(* Logix 5000 project; controller code_tcc vendor 1 type 14 code 106 rev 33.11; software revision 33.01; part 2 of 3 *)
(* tags used below, declared in another part *)
   Inp_Enable : BOOL;
   Ref_Connection : raC_UDT_ModbusClientConnection;
   Ref_Transactions : raC_UDT_ModbusClientTransaction[5];
   Ref_ModbusData : raC_UDT_ModbusClientData;
   Sts_Faulted : BOOL;
   Sts_Overlap : BOOL;
   Sts_Overload : BOOL;
   Wrk_MSGStep : DINT;
   Wrk_Main_Read_Buffer : STR4096;
   Wrk_WrIndex : DINT;
   Wrk_TransIndex : DINT;
   Wrk_TimerIndex : DINT;
   Wrk_ArraySize : DINT;
   Wrk_LastTransaction : DINT;
   Wrk_ClrReqIndex : DINT;
   Wrk_StepLockTimer : TIMER;
   Wrk_InitCompleted : BOOL;
   HMI_Tab : DINT;
   Wrk_tempHMItransaction : DINT;
   Wrk_HMITransactionValid : BOOL;
   wrk_FAL_Addr : CONTROL;
   wrk_LoopIndex : DINT;
   wrk_AddrIndex : DINT;
   HMI : raC_UDT_ModbusClientHMI;
   Wrk_OLindex : DINT;
   Wrk_OverloadStatus : BOOL;
   Wrk_OverlapStatus : BOOL;
(* raC_Opr_NetModbusTCPClient, continued *)

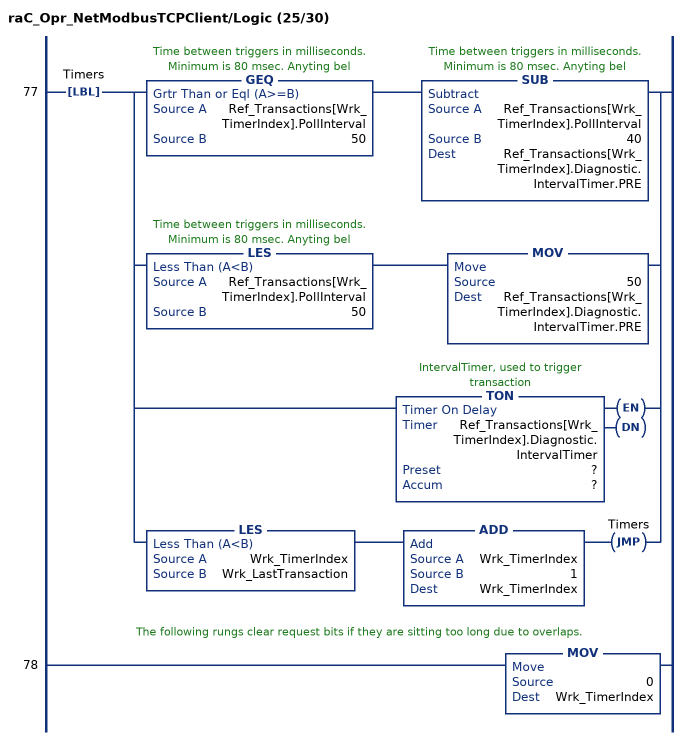
   77: LBL(Timers)[GEQ(Ref_Transactions[Wrk_TimerIndex].PollInterval,50) SUB(Ref_Transactions[Wrk_TimerIndex].PollInterval,40,Ref_Transactions[Wrk_TimerIndex].Diagnostic.IntervalTimer.PRE) ,LES(Ref_Transactions[Wrk_TimerIndex].PollInterval,50) MOV(50,Ref_Transactions[Wrk_TimerIndex].Diagnostic.IntervalTimer.PRE) ,TON(Ref_Transactions[Wrk_TimerIndex].Diagnostic.IntervalTimer,?,?) ,LES(Wrk_TimerIndex,Wrk_LastTransaction) ADD(Wrk_TimerIndex,1,Wrk_TimerIndex) JMP(Timers) ];
   // The following rungs clear request bits if they are sitting too long due to overlaps.
   78: MOV(0,Wrk_TimerIndex);
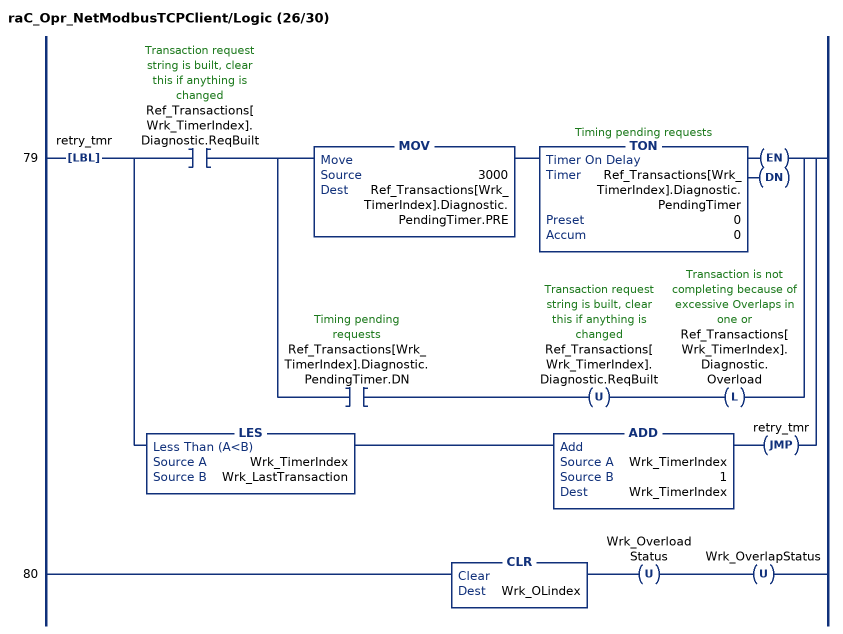
   79: LBL(retry_tmr)[XIC(Ref_Transactions[Wrk_TimerIndex].Diagnostic.ReqBuilt) [MOV(3000,Ref_Transactions[Wrk_TimerIndex].Diagnostic.PendingTimer.PRE) TON(Ref_Transactions[Wrk_TimerIndex].Diagnostic.PendingTimer,0,0) ,XIC(Ref_Transactions[Wrk_TimerIndex].Diagnostic.PendingTimer.DN) OTU(Ref_Transactions[Wrk_TimerIndex].Diagnostic.ReqBuilt) OTL(Ref_Transactions[Wrk_TimerIndex].Diagnostic.Overload) ] ,LES(Wrk_TimerIndex,Wrk_LastTransaction) ADD(Wrk_TimerIndex,1,Wrk_TimerIndex) JMP(retry_tmr) ];
   80: CLR(Wrk_OLindex)OTU(Wrk_OverloadStatus)OTU(Wrk_OverlapStatus);
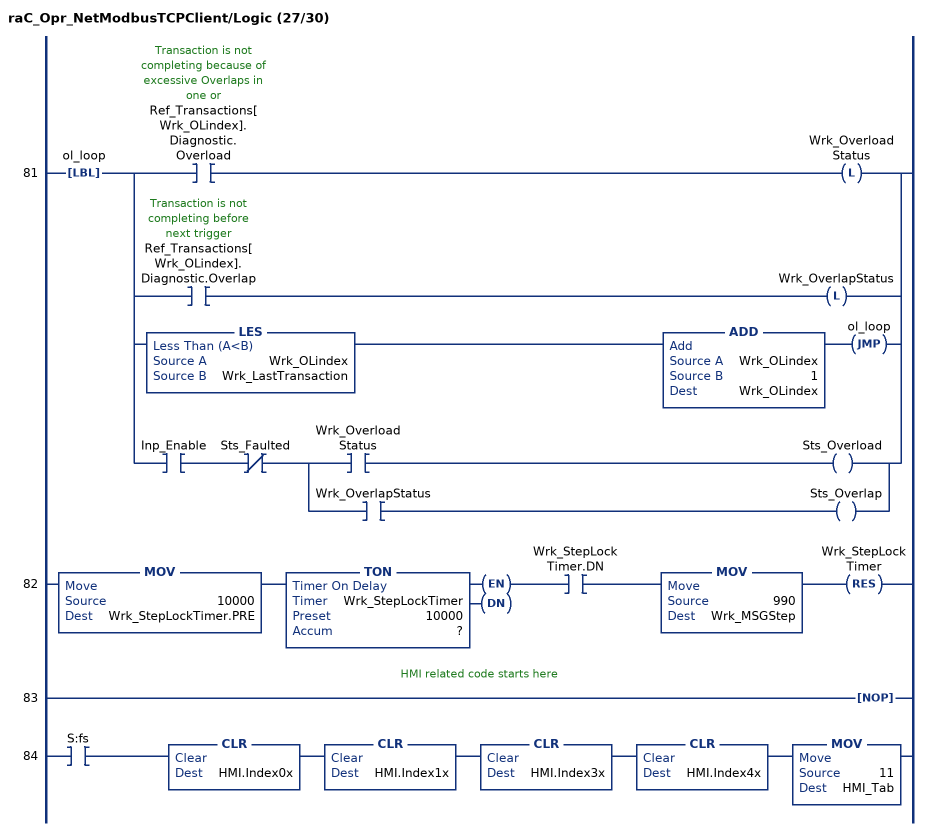
   81: LBL(ol_loop)[XIC(Ref_Transactions[Wrk_OLindex].Diagnostic.Overload) OTL(Wrk_OverloadStatus) ,XIC(Ref_Transactions[Wrk_OLindex].Diagnostic.Overlap) OTL(Wrk_OverlapStatus) ,LES(Wrk_OLindex,Wrk_LastTransaction) ADD(Wrk_OLindex,1,Wrk_OLindex) JMP(ol_loop) ,XIC(Inp_Enable) XIO(Sts_Faulted) [XIC(Wrk_OverloadStatus) OTE(Sts_Overload) ,XIC(Wrk_OverlapStatus) OTE(Sts_Overlap) ] ];
   82: MOV(10000,Wrk_StepLockTimer.PRE)TON(Wrk_StepLockTimer,?,?)XIC(Wrk_StepLockTimer.DN)MOV(990,Wrk_MSGStep)RES(Wrk_StepLockTimer);
   // HMI related code starts here
   83: NOP();
   84: XIC(S:fs)CLR(HMI.Index0x)CLR(HMI.Index1x)CLR(HMI.Index3x)CLR(HMI.Index4x)MOV(11,HMI_Tab);
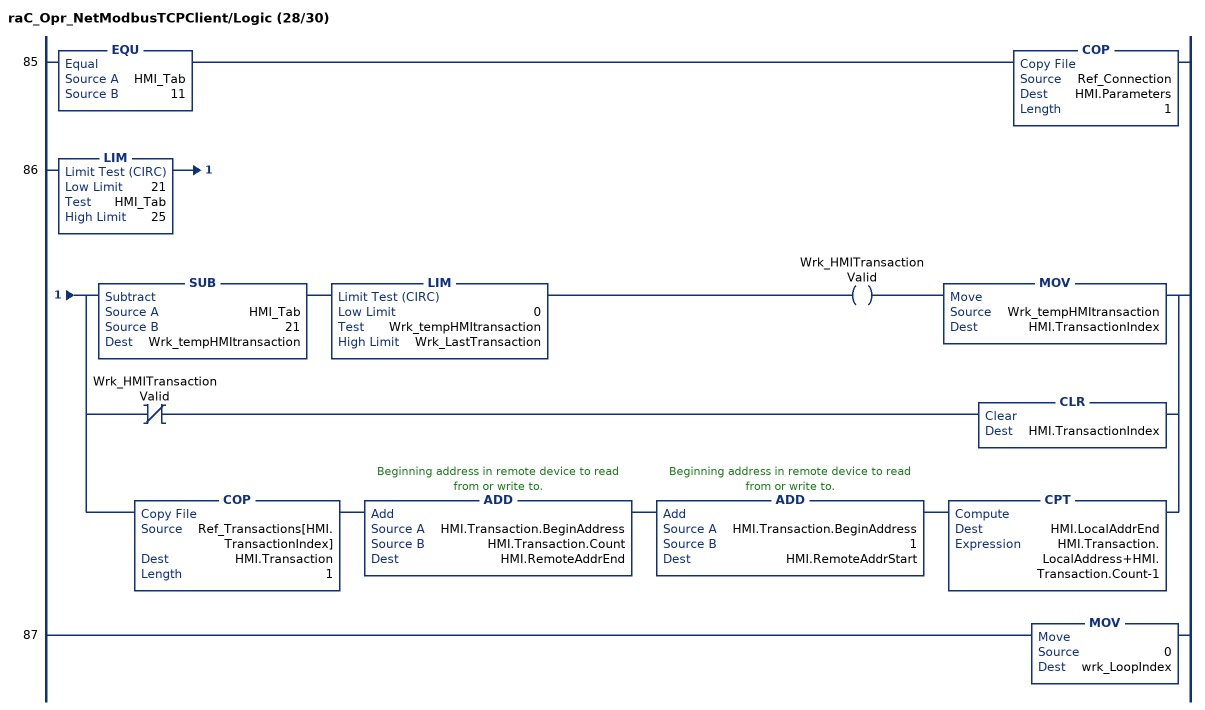
   85: EQU(HMI_Tab,11)COP(Ref_Connection,HMI.Parameters,1);
   86: LIM(21,HMI_Tab,25)[SUB(HMI_Tab,21,Wrk_tempHMItransaction) LIM(0,Wrk_tempHMItransaction,Wrk_LastTransaction) OTE(Wrk_HMITransactionValid) MOV(Wrk_tempHMItransaction,HMI.TransactionIndex) ,XIO(Wrk_HMITransactionValid) CLR(HMI.TransactionIndex) ,COP(Ref_Transactions[HMI.TransactionIndex],HMI.Transaction,1) ADD(HMI.Transaction.BeginAddress,HMI.Transaction.Count,HMI.RemoteAddrEnd) ADD(HMI.Transaction.BeginAddress,1,HMI.RemoteAddrStart) CPT(HMI.LocalAddrEnd,HMI.Transaction.LocalAddress+HMI.Transaction.Count-1) ];
   87: MOV(0,wrk_LoopIndex);
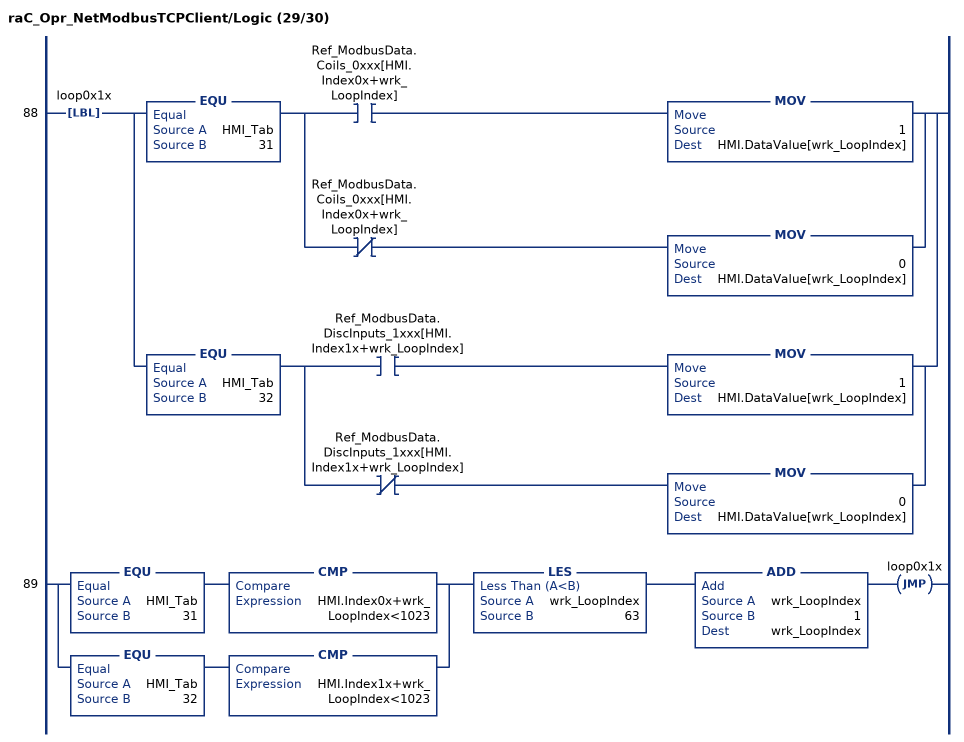
   88: LBL(loop0x1x)[EQU(HMI_Tab,31) [XIC(Ref_ModbusData.Coils_0xxx[HMI.Index0x+wrk_LoopIndex]) MOV(1,HMI.DataValue[wrk_LoopIndex]) ,XIO(Ref_ModbusData.Coils_0xxx[HMI.Index0x+wrk_LoopIndex]) MOV(0,HMI.DataValue[wrk_LoopIndex]) ] ,EQU(HMI_Tab,32) [XIC(Ref_ModbusData.DiscInputs_1xxx[HMI.Index1x+wrk_LoopIndex]) MOV(1,HMI.DataValue[wrk_LoopIndex]) ,XIO(Ref_ModbusData.DiscInputs_1xxx[HMI.Index1x+wrk_LoopIndex]) MOV(0,HMI.DataValue[wrk_LoopIndex]) ] ];
   89: [EQU(HMI_Tab,31) CMP(HMI.Index0x+wrk_LoopIndex<1023) ,EQU(HMI_Tab,32) CMP(HMI.Index1x+wrk_LoopIndex<1023) ]LES(wrk_LoopIndex,63)ADD(wrk_LoopIndex,1,wrk_LoopIndex)JMP(loop0x1x);
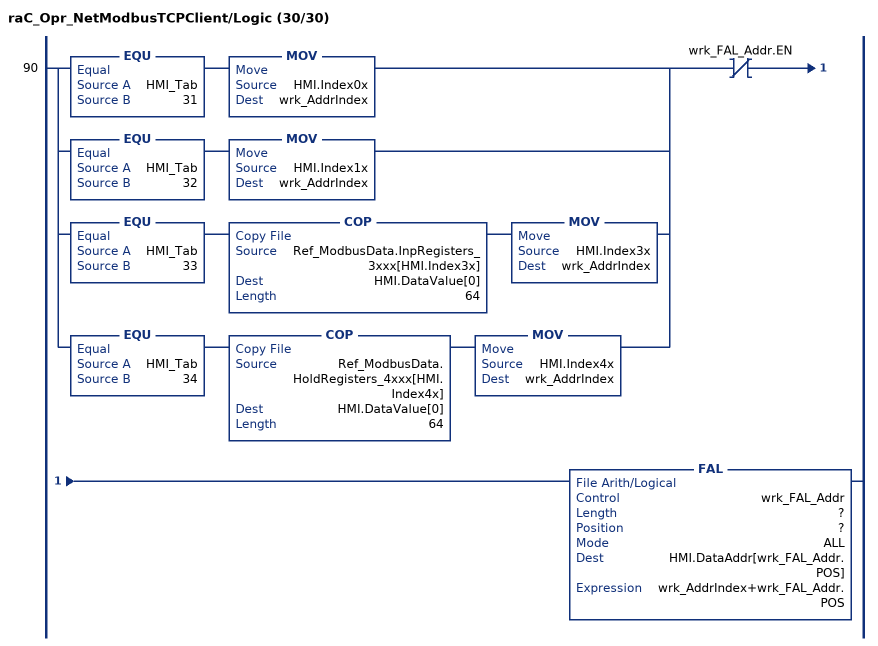
   90: [EQU(HMI_Tab,31) MOV(HMI.Index0x,wrk_AddrIndex) ,EQU(HMI_Tab,32) MOV(HMI.Index1x,wrk_AddrIndex) ,EQU(HMI_Tab,33) COP(Ref_ModbusData.InpRegisters_3xxx[HMI.Index3x],HMI.DataValue[0],64) MOV(HMI.Index3x,wrk_AddrIndex) ,EQU(HMI_Tab,34) COP(Ref_ModbusData.HoldRegisters_4xxx[HMI.Index4x],HMI.DataValue[0],64) MOV(HMI.Index4x,wrk_AddrIndex) ]XIO(wrk_FAL_Addr.EN)FAL(wrk_FAL_Addr,?,?,ALL,HMI.DataAddr[wrk_FAL_Addr.POS],wrk_AddrIndex+wrk_FAL_Addr.POS);
END_ROUTINE

ROUTINE Prescan   (* ladder *)
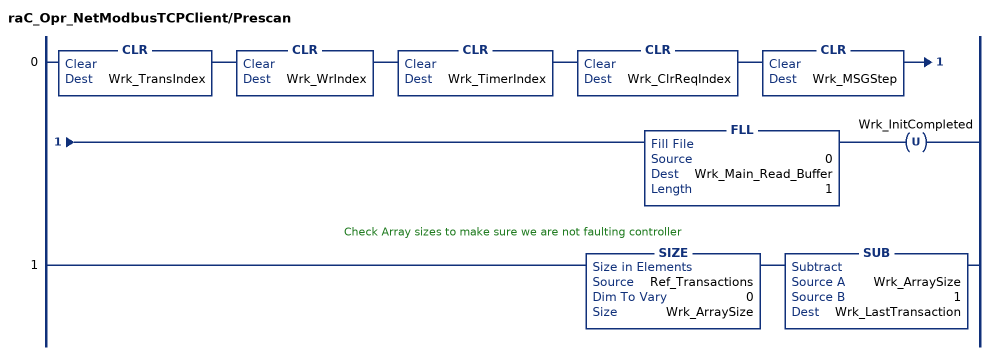
   0: CLR(Wrk_TransIndex)CLR(Wrk_WrIndex)CLR(Wrk_TimerIndex)CLR(Wrk_ClrReqIndex)CLR(Wrk_MSGStep)FLL(0,Wrk_Main_Read_Buffer,1)OTU(Wrk_InitCompleted);
   // Check Array sizes to make sure we are not faulting controller
   1: SIZE(Ref_Transactions,0,Wrk_ArraySize)SUB(Wrk_ArraySize,1,Wrk_LastTransaction);
END_ROUTINE
END_ADD_ON_INSTRUCTION

ADD_ON_INSTRUCTION raC_Tec_NetModbusTCPClient_BuildReqStr   (* revision 2.1, ExecutePrescan *)
// This routine builds a request string.
// Revision note:
// Moved to DINT in BeginAddress with boundary enforcement
VAR_IN_OUT
   Transaction : raC_UDT_ModbusClientTransaction; {required}
   ModbusData : raC_UDT_ModbusClientData; {required}
END_VAR
VAR_OUTPUT
   ER : BOOL; {access Read Only, visible}
END_VAR
VAR
   Wrk_TempInt : INT; {access None}
   Wrk_TempBeginInt : INT; {access None}
   Wrk_TempASCII_462 : STR0500; {access None}
   Wrk_Bit : DINT; {access None}
   Wrk_Byte : DINT; {access None}
   Wrk_Index : DINT; {access None}
   Wrk_LastAddr : DINT; {access None}
   Wrk_ValidRemoteRange : BOOL; {access None}
END_VAR

ROUTINE Logic   (* ladder *)
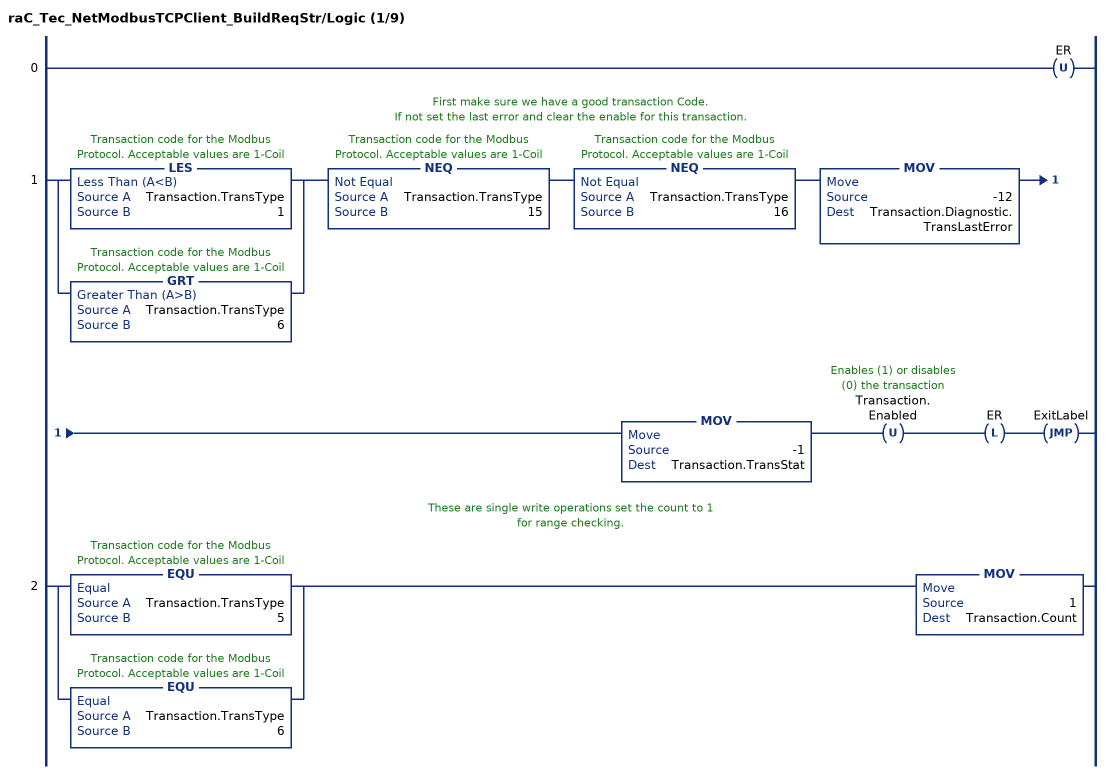
   0: OTU(ER);
   // First make sure we have a good transaction Code.
   // If not set the last error and clear the enable for this transaction.
   1: [LES(Transaction.TransType,1) ,GRT(Transaction.TransType,6) ]NEQ(Transaction.TransType,15)NEQ(Transaction.TransType,16)MOV(-12,Transaction.Diagnostic.TransLastError)MOV(-1,Transaction.TransStat)OTU(Transaction.Enabled)OTL(ER)JMP(ExitLabel);
   // These are single write operations set the count to 1
   //  for range checking.
   2: [EQU(Transaction.TransType,5) ,EQU(Transaction.TransType,6) ]MOV(1,Transaction.Count);
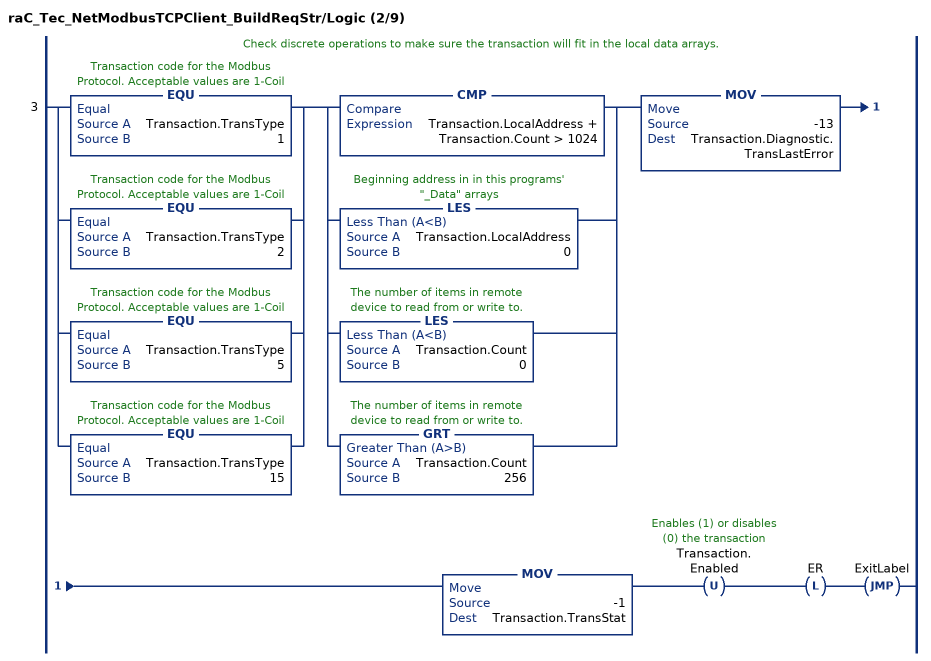
   // Check discrete operations to make sure the transaction will fit in the local data arrays.
   3: [EQU(Transaction.TransType,1) ,EQU(Transaction.TransType,2) ,EQU(Transaction.TransType,5) ,EQU(Transaction.TransType,15) ][CMP(Transaction.LocalAddress + Transaction.Count > 1024) ,LES(Transaction.LocalAddress,0) ,LES(Transaction.Count,0) ,GRT(Transaction.Count,256) ]MOV(-13,Transaction.Diagnostic.TransLastError)MOV(-1,Transaction.TransStat)OTU(Transaction.Enabled)OTL(ER)JMP(ExitLabel);
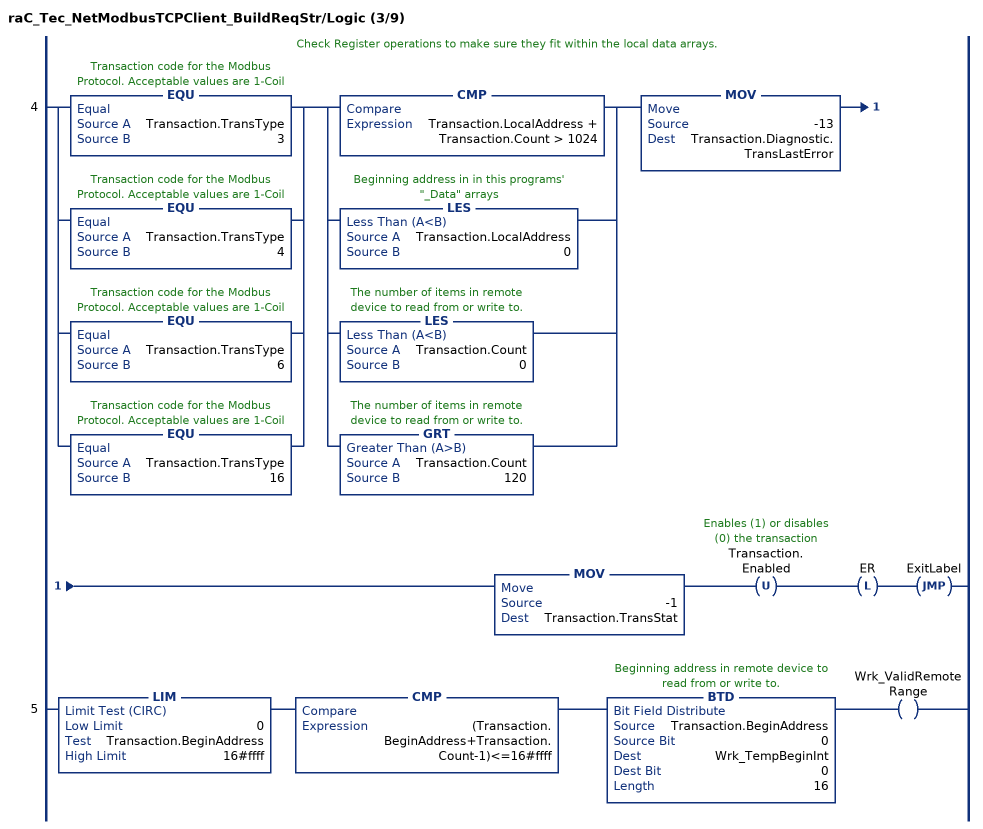
   // Check Register operations to make sure they fit within the local data arrays.
   4: [EQU(Transaction.TransType,3) ,EQU(Transaction.TransType,4) ,EQU(Transaction.TransType,6) ,EQU(Transaction.TransType,16) ][CMP(Transaction.LocalAddress + Transaction.Count > 1024) ,LES(Transaction.LocalAddress,0) ,LES(Transaction.Count,0) ,GRT(Transaction.Count,120) ]MOV(-13,Transaction.Diagnostic.TransLastError)MOV(-1,Transaction.TransStat)OTU(Transaction.Enabled)OTL(ER)JMP(ExitLabel);
   5: LIM(0,Transaction.BeginAddress,16#ffff)CMP((Transaction.BeginAddress+Transaction.Count-1)<=16#ffff)BTD(Transaction.BeginAddress,0,Wrk_TempBeginInt,0,16)OTE(Wrk_ValidRemoteRange);
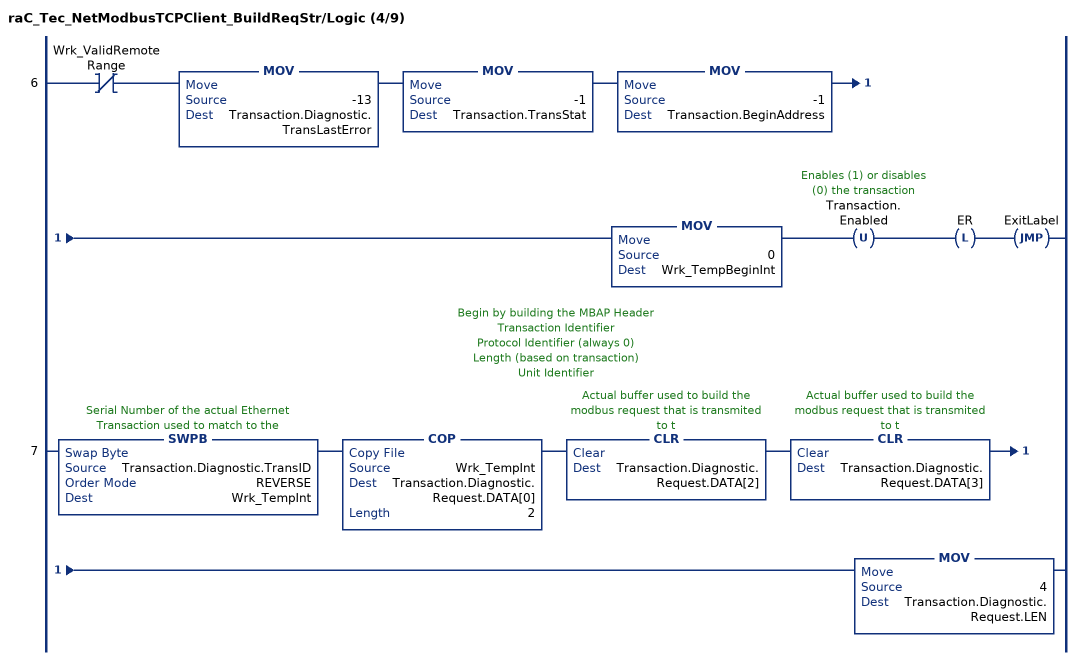
   6: XIO(Wrk_ValidRemoteRange)MOV(-13,Transaction.Diagnostic.TransLastError)MOV(-1,Transaction.TransStat)MOV(-1,Transaction.BeginAddress)MOV(0,Wrk_TempBeginInt)OTU(Transaction.Enabled)OTL(ER)JMP(ExitLabel);
   // Begin by building the MBAP Header
   // Transaction Identifier
   // Protocol Identifier (always 0)
   // Length (based on transaction)
   // Unit Identifier
   7: SWPB(Transaction.Diagnostic.TransID,REVERSE,Wrk_TempInt)COP(Wrk_TempInt,Transaction.Diagnostic.Request.DATA[0],2)CLR(Transaction.Diagnostic.Request.DATA[2])CLR(Transaction.Diagnostic.Request.DATA[3])MOV(4,Transaction.Diagnostic.Request.LEN);
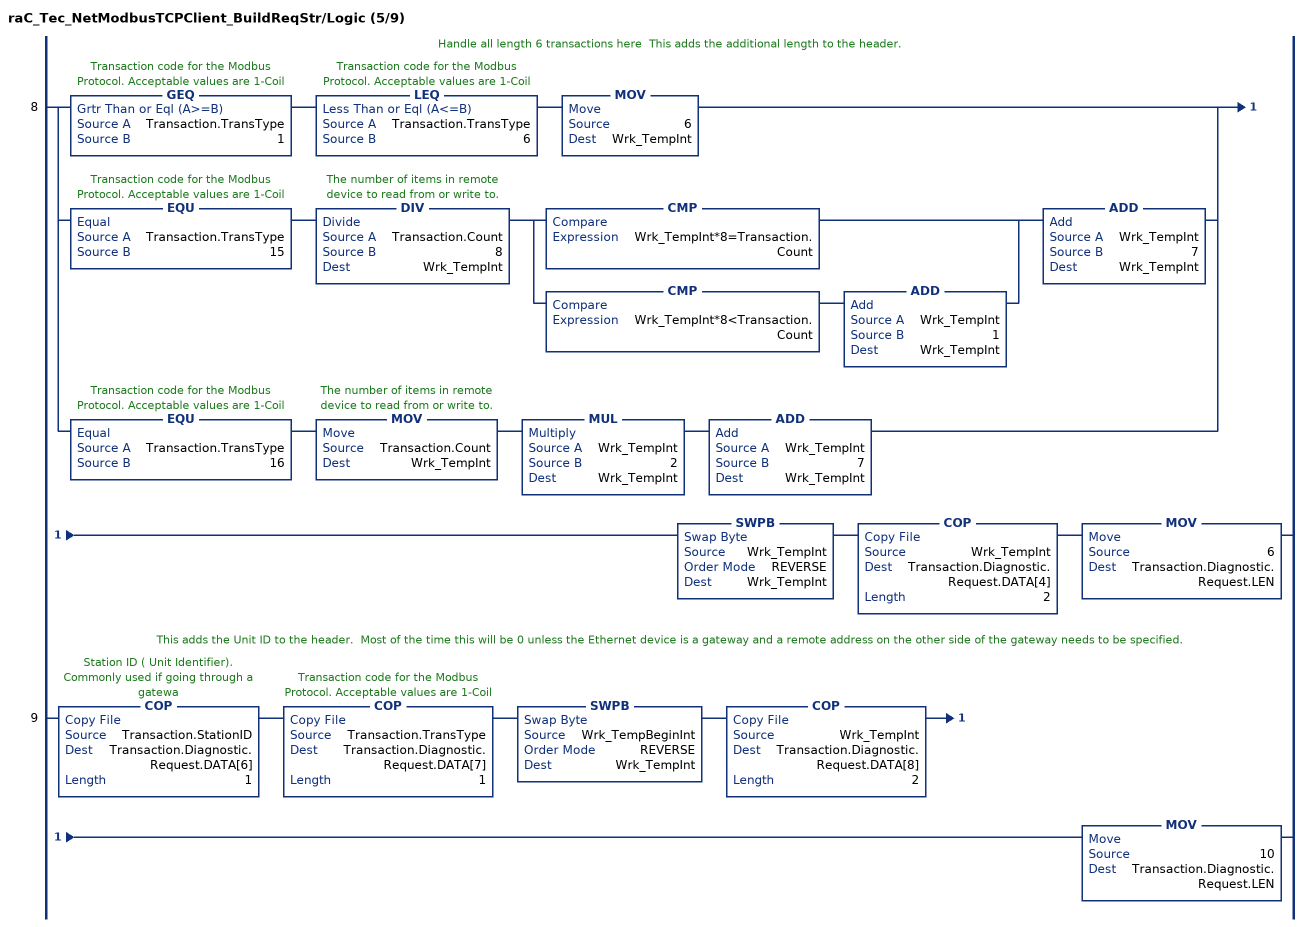
   // Handle all length 6 transactions here  This adds the additional length to the header.
   8: [GEQ(Transaction.TransType,1) LEQ(Transaction.TransType,6) MOV(6,Wrk_TempInt) ,EQU(Transaction.TransType,15) DIV(Transaction.Count,8,Wrk_TempInt) [CMP(Wrk_TempInt*8=Transaction.Count) ,CMP(Wrk_TempInt*8<Transaction.Count) ADD(Wrk_TempInt,1,Wrk_TempInt) ] ADD(Wrk_TempInt,7,Wrk_TempInt) ,EQU(Transaction.TransType,16) MOV(Transaction.Count,Wrk_TempInt) MUL(Wrk_TempInt,2,Wrk_TempInt) ADD(Wrk_TempInt,7,Wrk_TempInt) ]SWPB(Wrk_TempInt,REVERSE,Wrk_TempInt)COP(Wrk_TempInt,Transaction.Diagnostic.Request.DATA[4],2)MOV(6,Transaction.Diagnostic.Request.LEN);
   // This adds the Unit ID to the header.  Most of the time this will be 0 unless the Ethernet device is a gateway and a remote address on the other side of the gateway needs to be specified.
   9: COP(Transaction.StationID,Transaction.Diagnostic.Request.DATA[6],1)COP(Transaction.TransType,Transaction.Diagnostic.Request.DATA[7],1)SWPB(Wrk_TempBeginInt,REVERSE,Wrk_TempInt)COP(Wrk_TempInt,Transaction.Diagnostic.Request.DATA[8],2)MOV(10,Transaction.Diagnostic.Request.LEN);
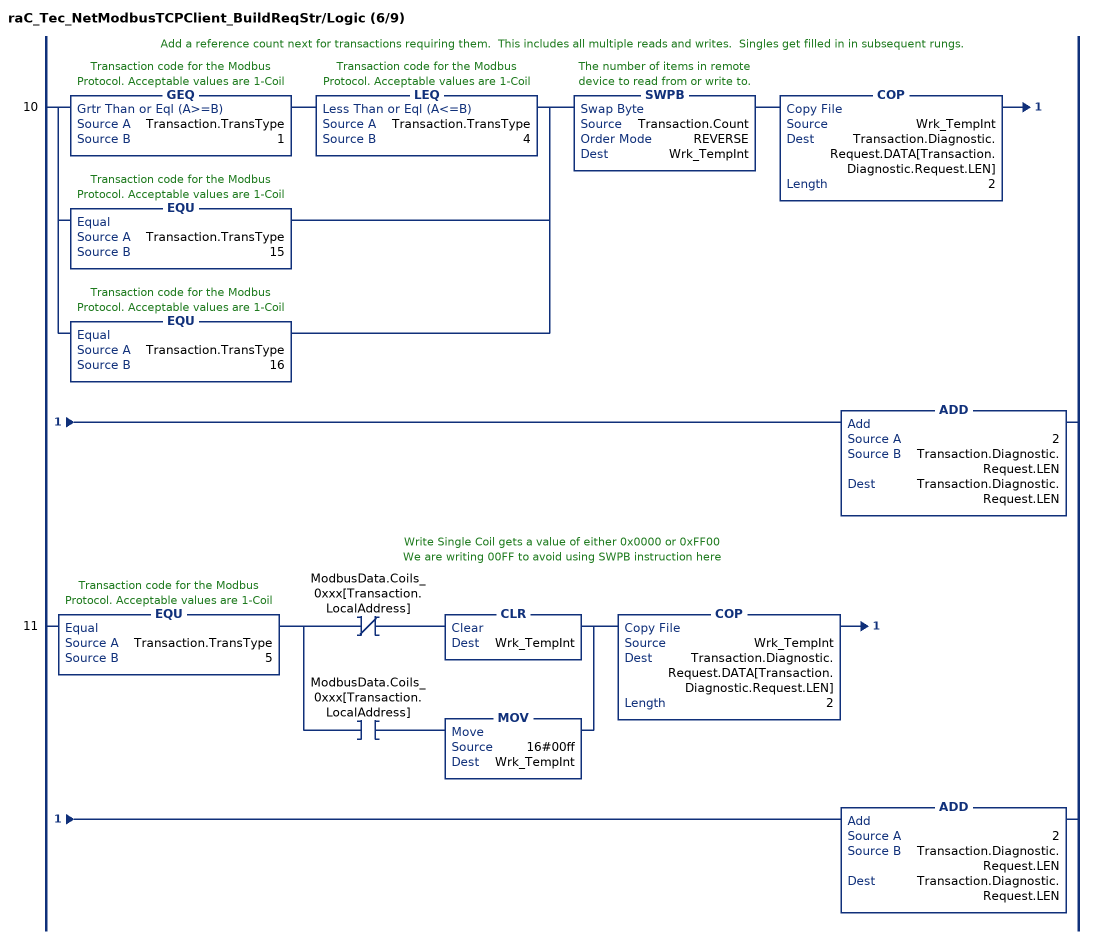
   // Add a reference count next for transactions requiring them.  This includes all multiple reads and writes.  Singles get filled in in subsequent rungs.
   10: [GEQ(Transaction.TransType,1) LEQ(Transaction.TransType,4) ,EQU(Transaction.TransType,15) ,EQU(Transaction.TransType,16) ]SWPB(Transaction.Count,REVERSE,Wrk_TempInt)COP(Wrk_TempInt,Transaction.Diagnostic.Request.DATA[Transaction.Diagnostic.Request.LEN],2)ADD(2,Transaction.Diagnostic.Request.LEN,Transaction.Diagnostic.Request.LEN);
   // Write Single Coil gets a value of either 0x0000 or 0xFF00
   // We are writing 00FF to avoid using SWPB instruction here
   11: EQU(Transaction.TransType,5)[XIO(ModbusData.Coils_0xxx[Transaction.LocalAddress]) CLR(Wrk_TempInt) ,XIC(ModbusData.Coils_0xxx[Transaction.LocalAddress]) MOV(16#00ff,Wrk_TempInt) ]COP(Wrk_TempInt,Transaction.Diagnostic.Request.DATA[Transaction.Diagnostic.Request.LEN],2)ADD(2,Transaction.Diagnostic.Request.LEN,Transaction.Diagnostic.Request.LEN);
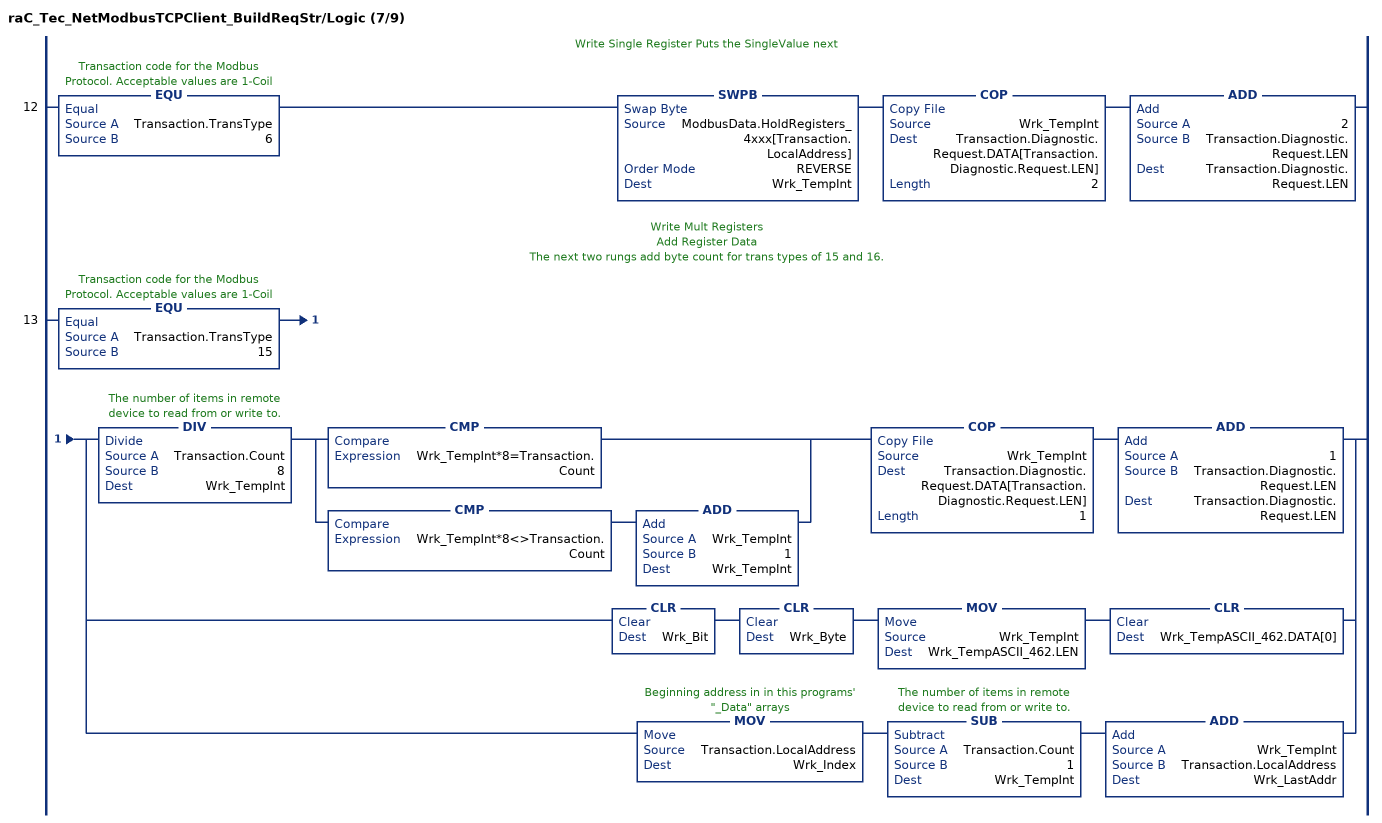
   // Write Single Register Puts the SingleValue next
   12: EQU(Transaction.TransType,6)SWPB(ModbusData.HoldRegisters_4xxx[Transaction.LocalAddress],REVERSE,Wrk_TempInt)COP(Wrk_TempInt,Transaction.Diagnostic.Request.DATA[Transaction.Diagnostic.Request.LEN],2)ADD(2,Transaction.Diagnostic.Request.LEN,Transaction.Diagnostic.Request.LEN);
   // Write Mult Registers
   // Add Register Data
   // The next two rungs add byte count for trans types of 15 and 16.
   13: EQU(Transaction.TransType,15)[DIV(Transaction.Count,8,Wrk_TempInt) [CMP(Wrk_TempInt*8=Transaction.Count) ,CMP(Wrk_TempInt*8<>Transaction.Count) ADD(Wrk_TempInt,1,Wrk_TempInt) ] COP(Wrk_TempInt,Transaction.Diagnostic.Request.DATA[Transaction.Diagnostic.Request.LEN],1) ADD(1,Transaction.Diagnostic.Request.LEN,Transaction.Diagnostic.Request.LEN) ,CLR(Wrk_Bit) CLR(Wrk_Byte) MOV(Wrk_TempInt,Wrk_TempASCII_462.LEN) CLR(Wrk_TempASCII_462.DATA[0]) ,MOV(Transaction.LocalAddress,Wrk_Index) SUB(Transaction.Count,1,Wrk_TempInt) ADD(Wrk_TempInt,Transaction.LocalAddress,Wrk_LastAddr) ];
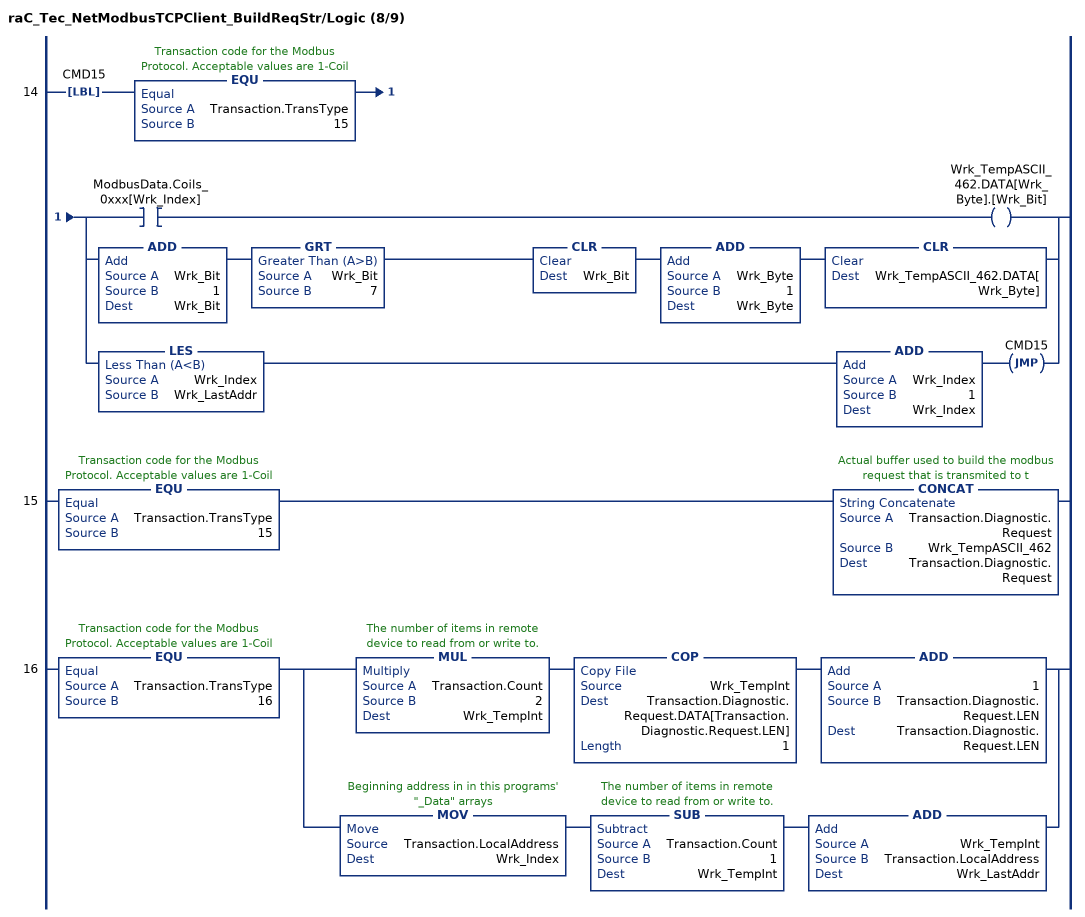
   14: LBL(CMD15)EQU(Transaction.TransType,15)[XIC(ModbusData.Coils_0xxx[Wrk_Index]) OTE(Wrk_TempASCII_462.DATA[Wrk_Byte].[Wrk_Bit]) ,ADD(Wrk_Bit,1,Wrk_Bit) GRT(Wrk_Bit,7) CLR(Wrk_Bit) ADD(Wrk_Byte,1,Wrk_Byte) CLR(Wrk_TempASCII_462.DATA[Wrk_Byte]) ,LES(Wrk_Index,Wrk_LastAddr) ADD(Wrk_Index,1,Wrk_Index) JMP(CMD15) ];
   15: EQU(Transaction.TransType,15)CONCAT(Transaction.Diagnostic.Request,Wrk_TempASCII_462,Transaction.Diagnostic.Request);
   16: EQU(Transaction.TransType,16)[MUL(Transaction.Count,2,Wrk_TempInt) COP(Wrk_TempInt,Transaction.Diagnostic.Request.DATA[Transaction.Diagnostic.Request.LEN],1) ADD(1,Transaction.Diagnostic.Request.LEN,Transaction.Diagnostic.Request.LEN) ,MOV(Transaction.LocalAddress,Wrk_Index) SUB(Transaction.Count,1,Wrk_TempInt) ADD(Wrk_TempInt,Transaction.LocalAddress,Wrk_LastAddr) ];
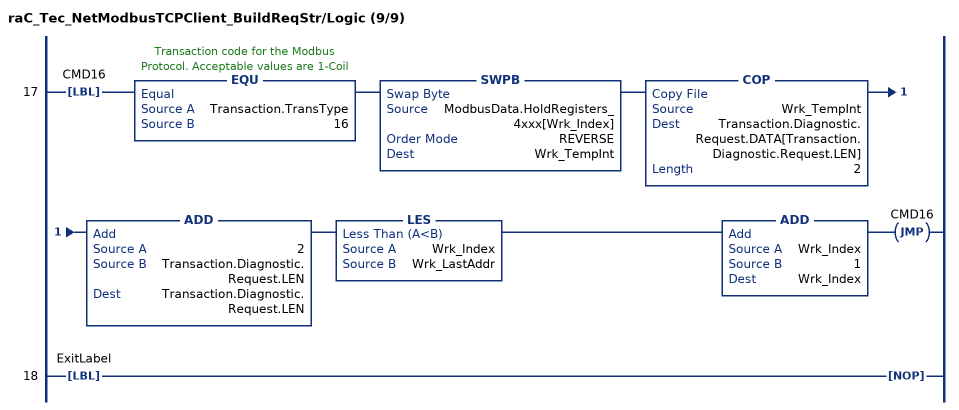
   17: LBL(CMD16)EQU(Transaction.TransType,16)SWPB(ModbusData.HoldRegisters_4xxx[Wrk_Index],REVERSE,Wrk_TempInt)COP(Wrk_TempInt,Transaction.Diagnostic.Request.DATA[Transaction.Diagnostic.Request.LEN],2)ADD(2,Transaction.Diagnostic.Request.LEN,Transaction.Diagnostic.Request.LEN)LES(Wrk_Index,Wrk_LastAddr)ADD(Wrk_Index,1,Wrk_Index)JMP(CMD16);
   18: LBL(ExitLabel)NOP();
END_ROUTINE

ROUTINE Prescan   (* ladder *)
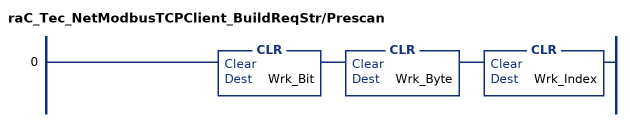
   0: CLR(Wrk_Bit)CLR(Wrk_Byte)CLR(Wrk_Index);
END_ROUTINE
END_ADD_ON_INSTRUCTION

ADD_ON_INSTRUCTION raC_Tec_NetModbusTCPClient_ChkWrReply   (* revision 2.0, ExecutePrescan *)
VAR_OUTPUT
   TransFound : BOOL; {access Read Only}
END_VAR
VAR_IN_OUT
   Transactions : raC_UDT_ModbusClientTransaction[5]; {required}
END_VAR
VAR_INPUT
   TransactionID : INT; {required}
   ModbusBytes : DINT; {required}
END_VAR
VAR_OUTPUT
   LocalOffset : INT; {access Read Only}
   Count : INT; {access Read Only}
END_VAR
VAR_INPUT
   Command : DINT; {required}
   LastTransaction : DINT; {required}
END_VAR
VAR
   Wrk_TransactionPtr : DINT; {access None}
END_VAR

ROUTINE Logic   (* ladder *)
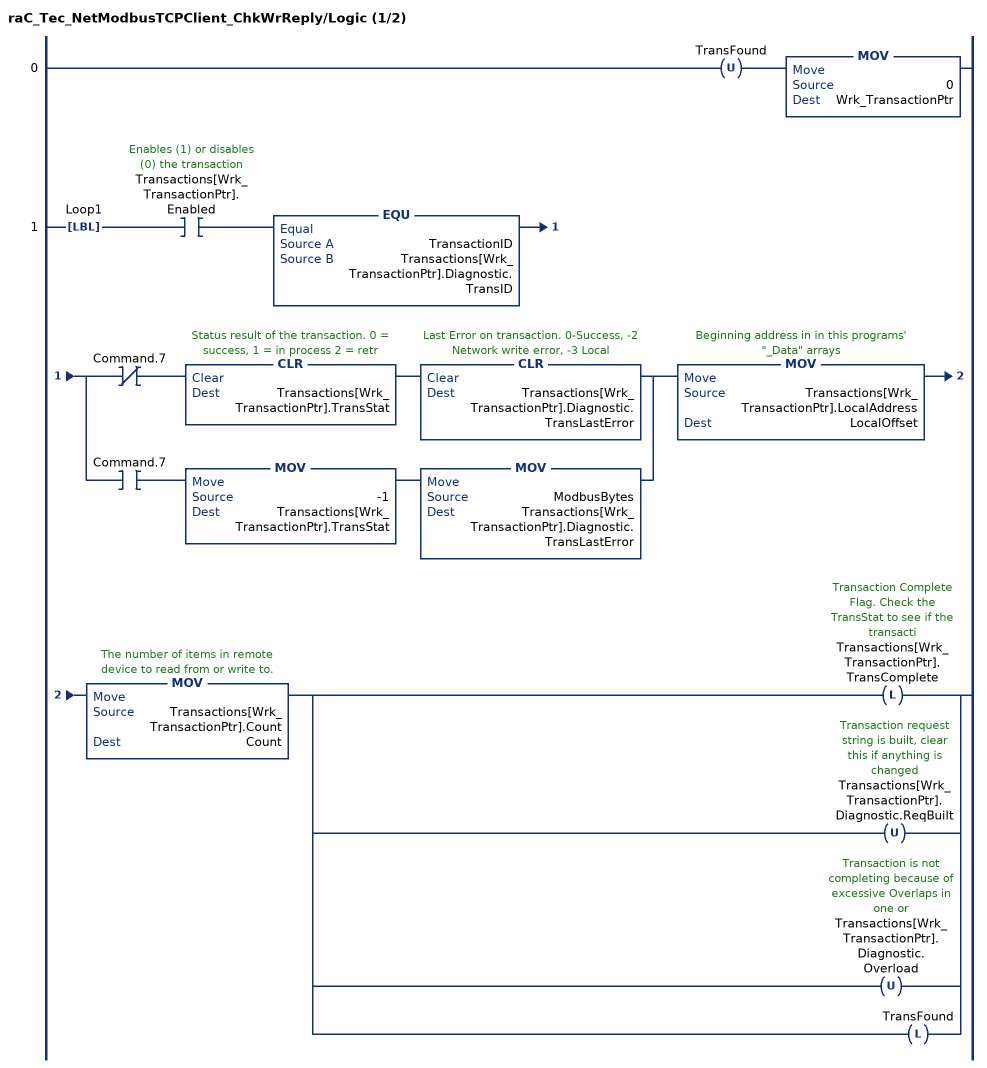
   0: OTU(TransFound)MOV(0,Wrk_TransactionPtr);
   1: LBL(Loop1)XIC(Transactions[Wrk_TransactionPtr].Enabled)EQU(TransactionID,Transactions[Wrk_TransactionPtr].Diagnostic.TransID)[XIO(Command.7) CLR(Transactions[Wrk_TransactionPtr].TransStat) CLR(Transactions[Wrk_TransactionPtr].Diagnostic.TransLastError) ,XIC(Command.7) MOV(-1,Transactions[Wrk_TransactionPtr].TransStat) MOV(ModbusBytes,Transactions[Wrk_TransactionPtr].Diagnostic.TransLastError) ]MOV(Transactions[Wrk_TransactionPtr].LocalAddress,LocalOffset)MOV(Transactions[Wrk_TransactionPtr].Count,Count)[OTL(Transactions[Wrk_TransactionPtr].TransComplete) ,OTU(Transactions[Wrk_TransactionPtr].Diagnostic.ReqBuilt) ,OTU(Transactions[Wrk_TransactionPtr].Diagnostic.Overload) ,OTL(TransFound) ];
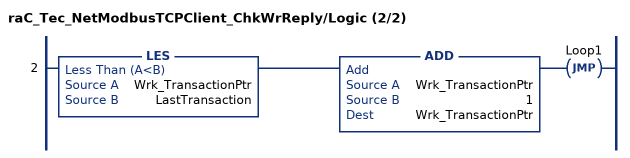
   2: LES(Wrk_TransactionPtr,LastTransaction)ADD(Wrk_TransactionPtr,1,Wrk_TransactionPtr)JMP(Loop1);
END_ROUTINE
